// TIA Portal V16 export
// export: Created 2022-02-28T20:45:45.6151989Z, ExportSetting WithDefaults, DisplayName Totally Integrated Automation Portal, DisplayVersion V16, DisplayName TIA Portal Version Control Interface, DisplayVersion V16, DisplayName TIA Portal Openness, DisplayVersion V16, DisplayName STEP 7 Professional, DisplayVersion V16, DisplayName STEP 7 Safety, DisplayVersion V16, DisplayName WinCC Advanced, DisplayVersion V16
FUNCTION_BLOCK "Modo_Auto-Manual"   // FB2, LAD
{ S7_Optimized_Access := 'TRUE' }
VERSION : 0.1
// stored: AutoNumber true, IsIECCheckEnabled false, IsRetainMemResEnabled false, MemoryReserve 100, SetENOAutomatically false, UDAEnableTagReadback false
   VAR_INPUT
      Confir_Perifericos : Bool;   // Confirmación Perifericos OK
      Modo_Automatico : Bool;
      Modo_Manual : Bool;
      Run_Btn : Bool;
      Stop_Btn : Bool;
      Run_HMI : Bool;
      Stop_HMI : Bool;
      Paro_Emergencia : Bool;
      "Remoto-Local" : Bool;
   END_VAR
   VAR_OUTPUT
      Arranque_Automatico : Bool;
      Arranque_Manual : Bool;
   END_VAR
   VAR
      Start_Remoto : Bool;
      Stop_Remoto : Bool;
   END_VAR
BEGIN

REGION Network 1: Modo Automático
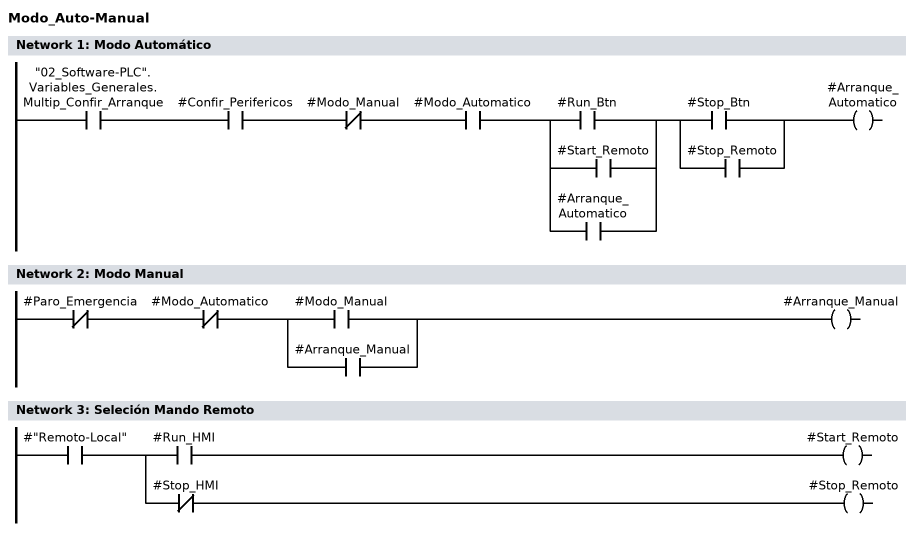
   RUNG wire#powerrail
      Contact( "02_Software-PLC".Variables_Generales.Multip_Confir_Arranque )
      Contact( #Confir_Perifericos )
      I_Contact( #Modo_Manual )
      Contact( #Modo_Automatico )
      wire#w1
      Contact( #Run_Btn )
      wire#w2
      Contact( #Stop_Btn )
      wire#w3
      Coil( #Arranque_Automatico )
   END_RUNG
   RUNG wire#w1
      Contact( #Start_Remoto )
   END_RUNG wire#w2
   RUNG wire#w1
      Contact( #Arranque_Automatico )
   END_RUNG wire#w2
   RUNG wire#w2
      Contact( #Stop_Remoto )
   END_RUNG wire#w3
   // the same network as SCL:
   #Arranque_Automatico := "02_Software-PLC".Variables_Generales.Multip_Confir_Arranque AND #Confir_Perifericos AND NOT #Modo_Manual AND #Modo_Automatico AND (#Run_Btn OR #Start_Remoto OR #Arranque_Automatico) AND (#Stop_Btn OR #Stop_Remoto);
END_REGION

REGION Network 2: Modo Manual
   RUNG wire#powerrail
      I_Contact( #Paro_Emergencia )
      I_Contact( #Modo_Automatico )
      wire#w1
      Contact( #Modo_Manual )
      wire#w2
      Coil( #Arranque_Manual )
   END_RUNG
   RUNG wire#w1
      Contact( #Arranque_Manual )
   END_RUNG wire#w2
   // the same network as SCL:
   #Arranque_Manual := NOT #Paro_Emergencia AND NOT #Modo_Automatico AND (#Modo_Manual OR #Arranque_Manual);
END_REGION

REGION Network 3: Seleción Mando Remoto
   RUNG wire#powerrail
      Contact( #"Remoto-Local" )
      wire#w1
      Contact( #Run_HMI )
      Coil( #Start_Remoto )
   END_RUNG
   RUNG wire#w1
      I_Contact( #Stop_HMI )
      Coil( #Stop_Remoto )
   END_RUNG
   // the same network as SCL:
   #Start_Remoto := #"Remoto-Local" AND #Run_HMI;
   #Stop_Remoto := #"Remoto-Local" AND NOT #Stop_HMI;
END_REGION
END_FUNCTION_BLOCK
